// TIA Portal V20 export
FUNCTION_BLOCK "SysFlipFlop"   // FB2000, FBD
TITLE = flip flop used for manual mode/push buttons
{ S7_Optimized_Access := 'TRUE' }
AUTHOR : MiCROTEC
VERSION : 1.0
// -2017.03 : Martin
// stored: AutoNumber false, MemoryReserve 100, SetENOAutomatically false
   VAR_INPUT
      input { ExternalAccessible := 'False'; ExternalVisible := 'False'; ExternalWritable := 'False'} : Bool;   // input toggle
      set { ExternalAccessible := 'False'; ExternalVisible := 'False'; ExternalWritable := 'False'} : Bool;   // set
      reset { ExternalAccessible := 'False'; ExternalVisible := 'False'; ExternalWritable := 'False'} : Bool;   // reset
      lmBlink { ExternalAccessible := 'False'; ExternalVisible := 'False'; ExternalWritable := 'False'} : Bool;   // let blink lamp
      lampTest { ExternalAccessible := 'False'; ExternalVisible := 'False'; ExternalWritable := 'False'} : Bool;   // lamp test
      resetMode { ExternalAccessible := 'False'; ExternalVisible := 'False'; ExternalWritable := 'False'} : Bool;   // 1=output will reset with rising edge from "LmBlink"
      hmiPageTar { ExternalAccessible := 'False'; ExternalVisible := 'False'; ExternalWritable := 'False'} : Int;   // number from hmi Page to open with rising edge from OutSignal
   END_VAR
   VAR_OUTPUT
      out { ExternalAccessible := 'False'; ExternalVisible := 'False'; ExternalWritable := 'False'} : Bool;   // output
      lamp { ExternalAccessible := 'False'; ExternalVisible := 'False'; ExternalWritable := 'False'} : Bool;   // lamp
      lamp2 { ExternalAccessible := 'False'; ExternalVisible := 'False'; ExternalWritable := 'False'} : Bool;   // lamp 2
      lamp3 { ExternalAccessible := 'False'; ExternalVisible := 'False'; ExternalWritable := 'False'} : Bool;   // lamp 3
   END_VAR
   VAR_IN_OUT
      hmiPageAct { ExternalAccessible := 'False'; ExternalVisible := 'False'; ExternalWritable := 'False'} : Int;
   END_VAR
   VAR RETAIN
      ff { ExternalAccessible := 'False'; ExternalVisible := 'False'; ExternalWritable := 'False'} : Bool;
      fl1 { ExternalAccessible := 'False'; ExternalVisible := 'False'; ExternalWritable := 'False'} : Bool;
      fl2 { ExternalAccessible := 'False'; ExternalVisible := 'False'; ExternalWritable := 'False'} : Bool;
      StatOut { ExternalAccessible := 'False'; ExternalVisible := 'False'; ExternalWritable := 'False'} : Bool;   // Setzen Rücksetzen über OP
   END_VAR
   VAR_TEMP   // added for the SCL form of the ladder/FBD networks
      _w1 : Bool;
   END_VAR
BEGIN

REGION Network 1: output
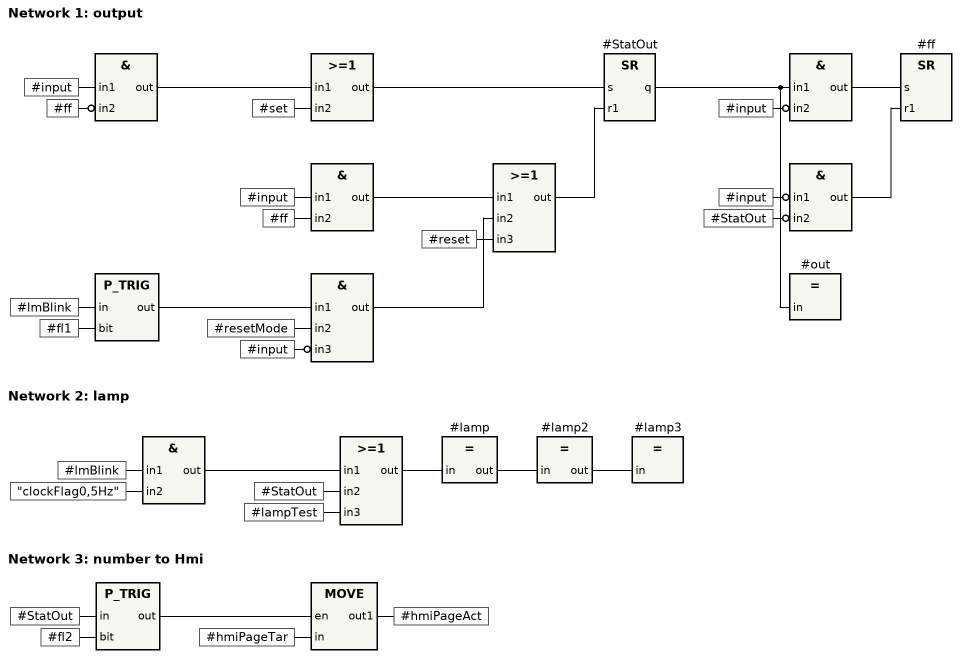
   #_w1 := #lmBlink AND NOT #fl1;   // rising edge
   #fl1 := #lmBlink;
   IF (#input AND NOT #ff) OR #set THEN
       #StatOut := TRUE;   // SR flip-flop
   END_IF;
   IF (#input AND #ff) OR (#_w1 AND #resetMode AND NOT #input) OR #reset THEN #StatOut := FALSE; END_IF;
   IF #StatOut AND NOT #input THEN
       #ff := TRUE;   // SR flip-flop
   END_IF;
   IF NOT #input AND NOT #StatOut THEN #ff := FALSE; END_IF;
   #out := #StatOut;
END_REGION

REGION Network 2: lamp
   #lamp := (#lmBlink AND "clockFlag0,5Hz") OR #StatOut OR #lampTest;
   #lamp2 := #lamp;
   #lamp3 := #lamp;
END_REGION

REGION Network 3: number to Hmi
   #_w1 := #StatOut AND NOT #fl2;   // rising edge
   #fl2 := #StatOut;
   IF #_w1 THEN #hmiPageAct := #hmiPageTar; END_IF;
END_REGION
END_FUNCTION_BLOCK
